// TIA Portal V18 export
ORGANIZATION_BLOCK "Main"   // OB1, LAD, ProgramCycle
TITLE = "Main Program Sweep (Cycle)"
{ S7_Optimized_Access := 'TRUE' }
VERSION : 0.1
// stored: AutoNumber true, IsIECCheckEnabled false, SetENOAutomatically false
BEGIN

REGION Network 1
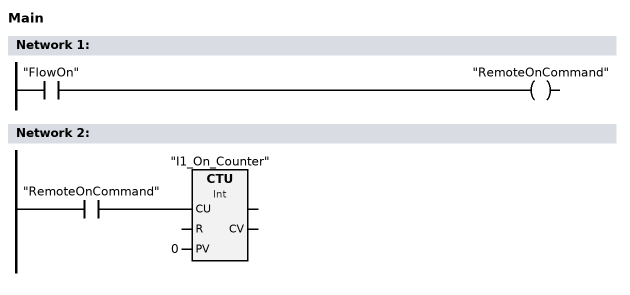
   RUNG wire#powerrail
      Contact( "FlowOn" )
      Coil( "RemoteOnCommand" )
   END_RUNG
   // the same network as SCL:
   "RemoteOnCommand" := "FlowOn";
END_REGION

REGION Network 2
   RUNG wire#powerrail
      Contact( "RemoteOnCommand" )
      { S7_Templates := "value_type := Int" } "I1_On_Counter".CTU(r :=, pv := 0, cv =>)
   END_RUNG
   // the same network as SCL:
   "I1_On_Counter".CTU(CU := "RemoteOnCommand", PV := 0);
END_REGION
END_ORGANIZATION_BLOCK
